FUNCTION_BLOCK FB_RecipeFactory
VAR
    BuilderWings 			: FB_PTPBorgoWings;
    BuilderFlaps 			: FB_PTPBorgoFlaps;
    BuilderArona 			: FB_PTPArona;
	BuilderRectangle 		: FB_PTPRectangle;
	
	BuilderCircle 			: FB_NCICircle;
	
	BuilderRoundedRect 		: FB_FeedRoundedRectangle;	
	BuilderFeedCircle  		: FB_FeedCircle;
	
	BuilderMeina2_2000x1000				: FB_FeedMeina2_2000x1000;
	BuilderMeina2_5Squares    			: FB_FeedMeina2_500x500;
    BuilderMeina2_500x500_Circles    	: FB_FeedMeina2_500x500_Circles;
    BuilderMeina2_3Squares    			: FB_FeedMeina2_750x750;
    BuilderMeina2_3Circles    			: FB_FeedMeina2_750x750_Circles;
    BuilderMeina2_1000x1000   			: FB_FeedMeina2_1000x1000;
    BuilderMeina2_1000x1000_Circles    	: FB_FeedMeina2_1000x1000_Circles;
    BuilderMeina2_2000x500    			: FB_FeedMeina2_2000x500;
	
	BuilderMeina2_Samples				: FB_FeedMeina2_Samples;
END_VAR

METHOD GetBuilder : I_RecipeBuilder
VAR_INPUT
    RequestedRecipe : E_RecipeID;
END_VAR
CASE RequestedRecipe OF
    E_RecipeID.ePTPBorgoWings:
        GetBuilder := BuilderWings; 
        
    E_RecipeID.ePTPBorgoFlaps:
        GetBuilder := BuilderFlaps;
        
    E_RecipeID.ePTPArona:
        GetBuilder := BuilderArona;
		
	E_RecipeID.eNCICircle:
        GetBuilder := BuilderCircle;
		
	E_RecipeID.ePTPRectangle:                            
        GetBuilder := BuilderRectangle; 
	
	E_RecipeID.eFeedRoundedRectangle:                            
        GetBuilder := BuilderRoundedRect;    

	E_RecipeID.eFeedCircle:                 
        GetBuilder := BuilderFeedCircle;        

	E_RecipeID.eFeedMeina2_2000x1000:
		GetBuilder := BuilderMeina2_2000x1000;   
		
	E_RecipeID.eFeedMeina2_500x500:    
		GetBuilder := BuilderMeina2_5Squares;
		
    E_RecipeID.eFeedMeina2_500x500_Circles:    
		GetBuilder := BuilderMeina2_500x500_Circles;
		
    E_RecipeID.eFeedMeina2_750x750:    
		GetBuilder := BuilderMeina2_3Squares;
		
    E_RecipeID.eFeedMeina2_750x750_Circles:    
		GetBuilder := BuilderMeina2_3Circles;
		
    E_RecipeID.eFeedMeina2_1000x1000:    
		GetBuilder := BuilderMeina2_1000x1000;
		
    E_RecipeID.eFeedMeina2_1000x1000_Circles:    
		GetBuilder := BuilderMeina2_1000x1000_Circles;
		
    E_RecipeID.eFeedMeina2_2000x500: 
		GetBuilder := BuilderMeina2_2000x500;
		
	E_RecipeID.eFeedMeina2_Samples: 
		GetBuilder := BuilderMeina2_Samples;	
        
ELSE
    GetBuilder := 0; 
END_CASE
END_METHOD

METHOD InitializeFactory
VAR_INPUT
    Config : ST_RecipeBuilder_Config;
	ConfigProvider : I_GantryConfigProvider;
END_VAR
BuilderWings.Config 				:= Config;
BuilderWings.ConfigProvider 		:= ConfigProvider; 

BuilderFlaps.Config 				:= Config;
BuilderFlaps.ConfigProvider 		:= ConfigProvider;

BuilderArona.Config 				:= Config;
BuilderArona.ConfigProvider 		:= ConfigProvider;

BuilderCircle.Config 				:= Config;
BuilderCircle.ConfigProvider 		:= ConfigProvider;

BuilderRectangle.Config 			:= Config;                    
BuilderRectangle.ConfigProvider 	:= ConfigProvider; 
   
BuilderRoundedRect.Config 			:= Config;
BuilderRoundedRect.ConfigProvider 	:= ConfigProvider;

BuilderFeedCircle.Config 			:= Config;                    
BuilderFeedCircle.ConfigProvider 	:= ConfigProvider;

BuilderMeina2_2000x1000.Config				:= Config;    
BuilderMeina2_2000x1000.ConfigProvider		:= ConfigProvider;

BuilderMeina2_5Squares.Config       := Config;
BuilderMeina2_5Squares.ConfigProvider := ConfigProvider;

BuilderMeina2_500x500_Circles.Config       := Config;
BuilderMeina2_500x500_Circles.ConfigProvider := ConfigProvider;

BuilderMeina2_3Squares.Config       := Config;
BuilderMeina2_3Squares.ConfigProvider := ConfigProvider;

BuilderMeina2_3Circles.Config       := Config;
BuilderMeina2_3Circles.ConfigProvider := ConfigProvider;

BuilderMeina2_1000x1000.Config       := Config;
BuilderMeina2_1000x1000.ConfigProvider := ConfigProvider;

BuilderMeina2_1000x1000_Circles.Config       := Config;
BuilderMeina2_1000x1000_Circles.ConfigProvider := ConfigProvider;

BuilderMeina2_2000x500.Config    := Config;
BuilderMeina2_2000x500.ConfigProvider := ConfigProvider;    

BuilderMeina2_Samples.Config    := Config;
BuilderMeina2_Samples.ConfigProvider := ConfigProvider;
END_METHOD

METHOD UpdateConfig
VAR_INPUT
    Config : ST_RecipeBuilder_Config;
END_VAR
// Fabryka rozsyła nową konfigurację do wszystkich swoich "dzieci"
BuilderWings.Config 		:= Config;
BuilderFlaps.Config 		:= Config;
BuilderArona.Config 		:= Config;
BuilderCircle.Config 		:= Config;
BuilderRectangle.Config 	:= Config;   
BuilderRoundedRect.Config 	:= Config;      
BuilderFeedCircle.Config 	:= Config; 
BuilderMeina2_2000x1000.Config		:= Config;                 
BuilderMeina2_5Squares.Config    := Config;
BuilderMeina2_500x500_Circles.Config    := Config;
BuilderMeina2_3Squares.Config    := Config;
BuilderMeina2_3Circles.Config    := Config;
BuilderMeina2_1000x1000.Config    := Config;
BuilderMeina2_1000x1000_Circles.Config    := Config;
BuilderMeina2_2000x500.Config := Config;
BuilderMeina2_Samples.Config := Config;
END_METHOD

END_FUNCTION_BLOCK

(* stored: Version 1.1.0.1, ProductVersion 3.1.4024.15
   POU FB_RecipeFactory: Id {eb67f754-8d88-44c2-acf6-733dd105dd46}, SpecialFunc None
   Method GetBuilder: Id {4ef94639-3187-4b95-bdcd-c7a9da21c9f0}
   Method InitializeFactory: Id {d617016c-6308-411a-9cc3-c9f77798a181}
   Method UpdateConfig: Id {addb126c-7b31-4fe1-bab5-a92c30ad08f7} *)
